(* Logix 5000 project; controller VET 1756-L62 rev 19.52; software revision 19.01; part 18 of 27 *)
(* tags used below, declared in another part *)
   dosif_struct : ALIAS FOR dosificador[1];
   dosificacion_interrumpida : BOOL;
   dosificando : BOOL;
   flags : DINT;
   idx_batch : DINT;
   idx_eqp1 : DINT;
   idx_eqp2 : DINT;
   idx_eqp3 : DINT;
   idx_eqp4 : DINT;
   idx_eqp5 : DINT;
   idx_ing : DINT;
   idx_tolv : DINT;   // Índice de Tolva
   resultado : ALIAS FOR dosif_struct.resultado;
   step_index : DINT;
   step_index_buffer : DINT;
   T : TIMER[15];
   _Eqp : Equipo[800];
   _Parametros_D : DINT[30];
   _Parametros_F : REAL[30];
   _reset_locales : DINT;
   Batch : batch[10];
   corriente : REAL[40];
   dosificador : dosif_struct[20];
   Dosificar_MID_01 : PHASE;
   fecha_plc : DINT;
   flujometro : flujometro[5];
   hora_plc : DINT;
   peso_tolva : REAL[80];
   SetDInt : DINT[500];
   TabBin : Bins_Setup;
   vdf : VDFS[20];
(* Dosificar_MID_01, continued *)

ROUTINE Holding   (* ladder *)
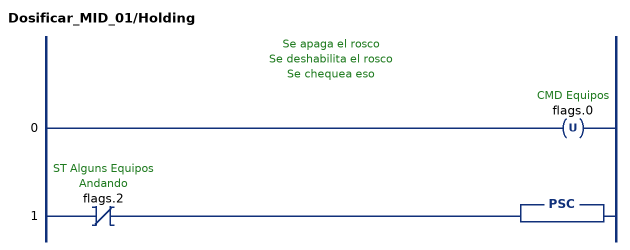
   // Se apaga el rosco
   // Se deshabilita el rosco
   // Se chequea eso
   0: OTU(flags.0);
   1: XIO(flags.2)PSC();
END_ROUTINE

ROUTINE preState   (* ladder *)
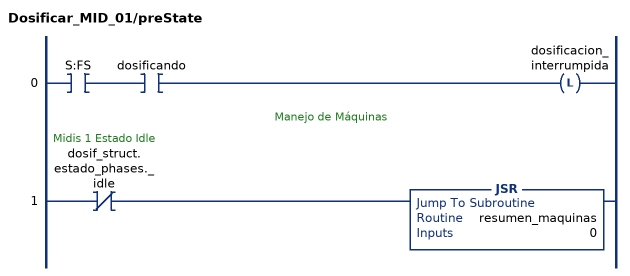
   0: XIC(S:FS)XIC(dosificando)OTL(dosificacion_interrumpida);
   // Manejo de Máquinas
   1: XIO(dosif_struct.estado_phases._idle)JSR(resumen_maquinas,0);
END_ROUTINE

ROUTINE Resetting   (* ladder *)
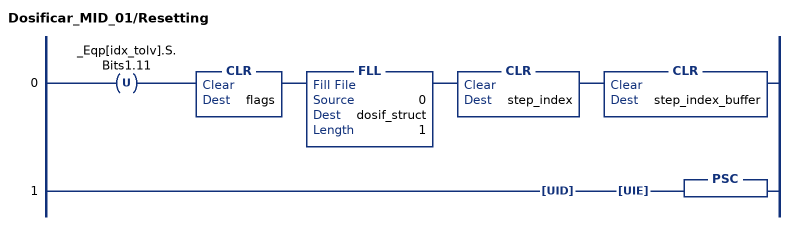
   0: OTU(_Eqp[idx_tolv].S.Bits1.11)CLR(flags)FLL(0,dosif_struct,1)CLR(step_index)CLR(step_index_buffer);
   1: UID()UIE()PSC();
END_ROUTINE

ROUTINE Restarting   (* ladder *)
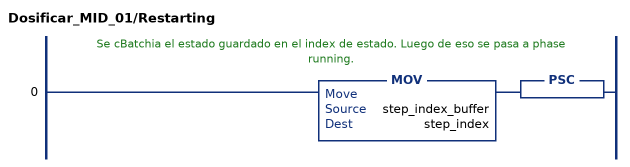
   // Se cBatchia el estado guardado en el index de estado. Luego de eso se pasa a phase running.
   0: MOV(step_index_buffer,step_index)PSC();
END_ROUTINE

ROUTINE resumen_maquinas   (* ladder *)
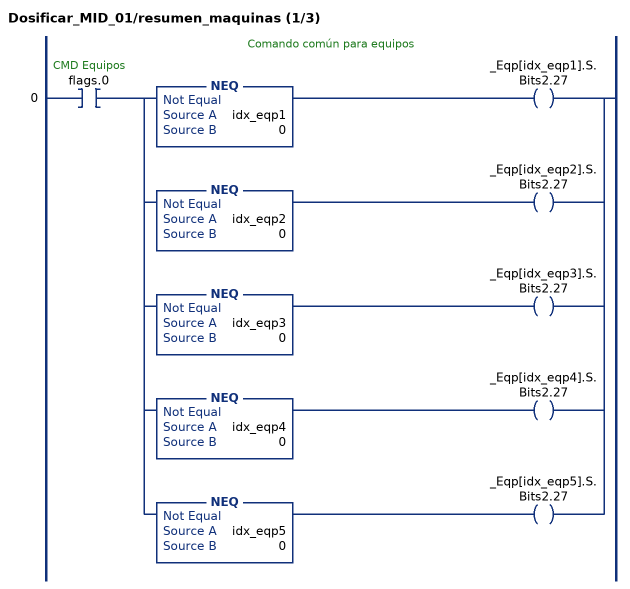
   // Comando común para equipos
   0: XIC(flags.0)[NEQ(idx_eqp1,0) OTE(_Eqp[idx_eqp1].S.Bits2.27) ,NEQ(idx_eqp2,0) OTE(_Eqp[idx_eqp2].S.Bits2.27) ,NEQ(idx_eqp3,0) OTE(_Eqp[idx_eqp3].S.Bits2.27) ,NEQ(idx_eqp4,0) OTE(_Eqp[idx_eqp4].S.Bits2.27) ,NEQ(idx_eqp5,0) OTE(_Eqp[idx_eqp5].S.Bits2.27) ];
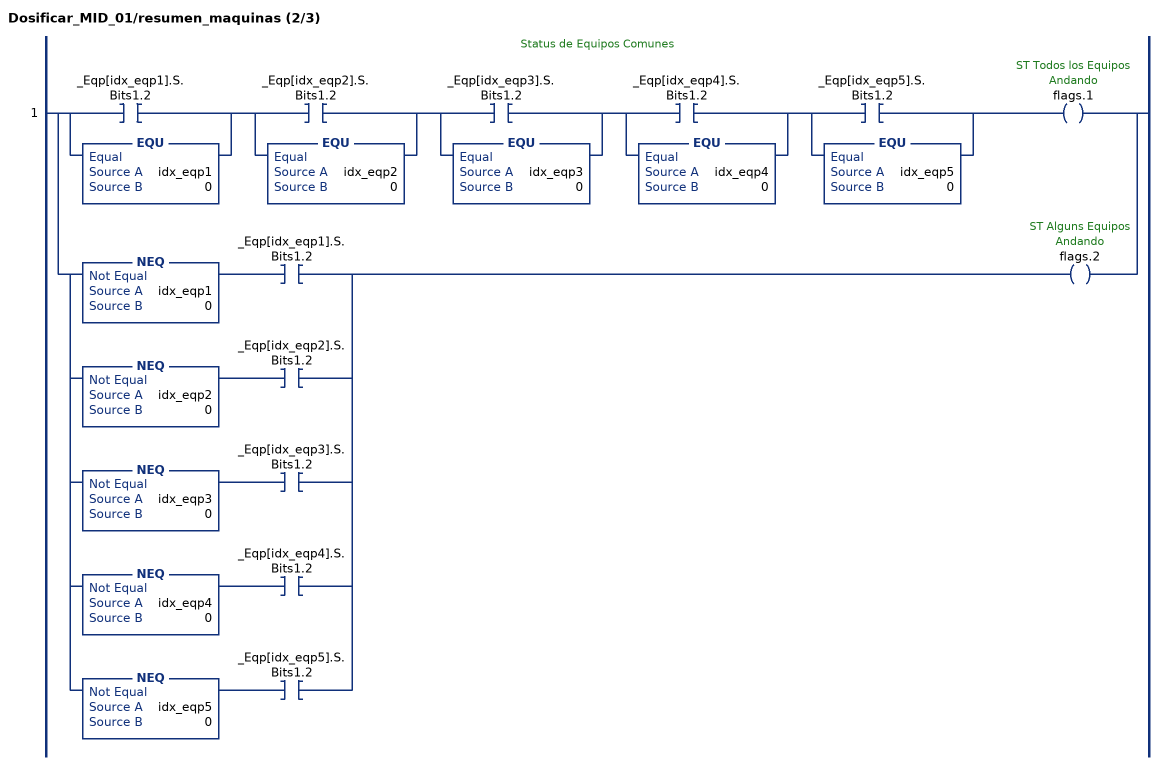
   // Status de Equipos Comunes
   1: [[XIC(_Eqp[idx_eqp1].S.Bits1.2) ,EQU(idx_eqp1,0) ] [XIC(_Eqp[idx_eqp2].S.Bits1.2) ,EQU(idx_eqp2,0) ] [XIC(_Eqp[idx_eqp3].S.Bits1.2) ,EQU(idx_eqp3,0) ] [XIC(_Eqp[idx_eqp4].S.Bits1.2) ,EQU(idx_eqp4,0) ] [XIC(_Eqp[idx_eqp5].S.Bits1.2) ,EQU(idx_eqp5,0) ] OTE(flags.1) ,[NEQ(idx_eqp1,0) XIC(_Eqp[idx_eqp1].S.Bits1.2) ,NEQ(idx_eqp2,0) XIC(_Eqp[idx_eqp2].S.Bits1.2) ,NEQ(idx_eqp3,0) XIC(_Eqp[idx_eqp3].S.Bits1.2) ,NEQ(idx_eqp4,0) XIC(_Eqp[idx_eqp4].S.Bits1.2) ,NEQ(idx_eqp5,0) XIC(_Eqp[idx_eqp5].S.Bits1.2) ] OTE(flags.2) ];
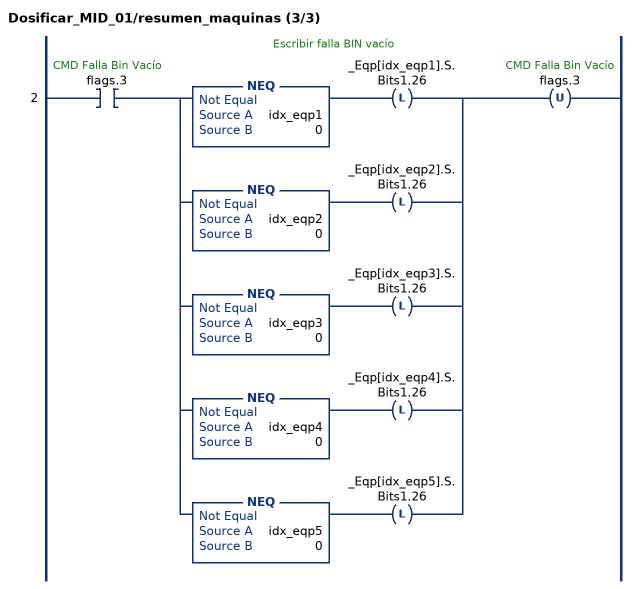
   // Escribir falla BIN vacío
   2: XIC(flags.3)[NEQ(idx_eqp1,0) OTL(_Eqp[idx_eqp1].S.Bits1.26) ,NEQ(idx_eqp2,0) OTL(_Eqp[idx_eqp2].S.Bits1.26) ,NEQ(idx_eqp3,0) OTL(_Eqp[idx_eqp3].S.Bits1.26) ,NEQ(idx_eqp4,0) OTL(_Eqp[idx_eqp4].S.Bits1.26) ,NEQ(idx_eqp5,0) OTL(_Eqp[idx_eqp5].S.Bits1.26) ]OTU(flags.3);
END_ROUTINE

ROUTINE Running   (* ladder *)
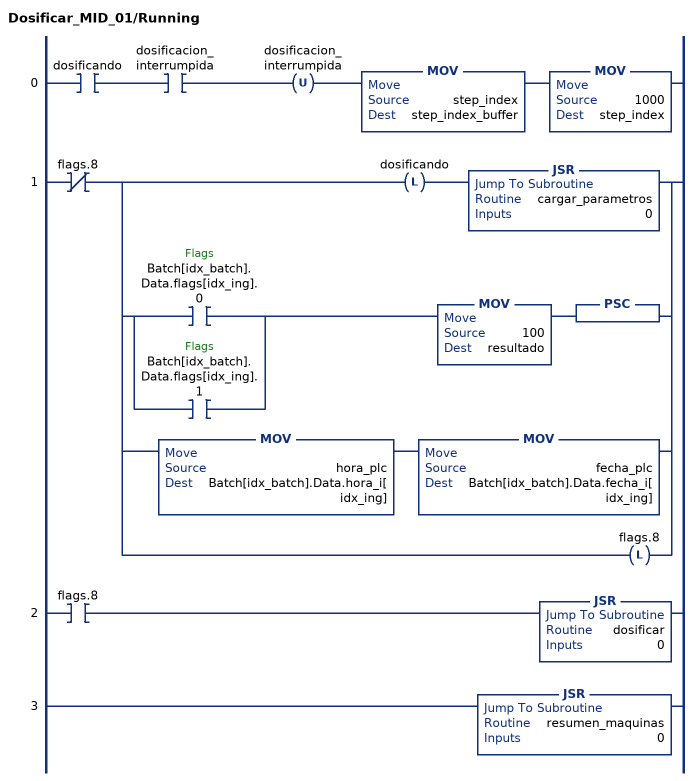
   0: XIC(dosificando)XIC(dosificacion_interrumpida)OTU(dosificacion_interrumpida)MOV(step_index,step_index_buffer)MOV(1000,step_index);
   1: XIO(flags.8)[OTL(dosificando) JSR(cargar_parametros,0) ,[[XIC(Batch[idx_batch].Data.flags[idx_ing].0) ,XIC(Batch[idx_batch].Data.flags[idx_ing].1) ] MOV(100,resultado) PSC() ,MOV(hora_plc,Batch[idx_batch].Data.hora_i[idx_ing]) MOV(fecha_plc,Batch[idx_batch].Data.fecha_i[idx_ing]) ] ,OTL(flags.8) ];
   2: XIC(flags.8)JSR(dosificar,0);
   3: JSR(resumen_maquinas,0);
END_ROUTINE
END_PROGRAM

PROGRAM Gestion_Dosificacion   (* main routine Main *)
VAR
   _fn1_auto : BOOL := 1;
   _fn1_ingrediente : DINT := 66;
   _fn1_lugar : DINT := 2;
   _fn1_ndx : DINT := 42;
   _fn1_prioridad : DINT;
   _fn1_tolva : DINT[2] := ([0] := 17);
   _fn2_batch_detalle : batch_detalle := (codigo[0] := 81, codigo[1] := 51, codigo[2] := 53, codigo[3] := 55, codigo[4] := 57, codigo[5] := 67, codigo[6] := 68, codigo[7] := 69, codigo[8] := 70, codigo[9] := 74, codigo[10] := 75, codigo[11] := 76, codigo[12] := 77, codigo[13] := 60, codigo[14] := 62, codigo[15] := 64, codigo[16] := 66, peso_f[0] := 70.0, peso_f[1] := 400.0, peso_f[2] := 350.0, peso_f[3] := 175.0, peso_f[4] := 225.0, peso_f[5] := 30.0, peso_f[6] := 25.0, peso_f[7] := 17.5, peso_f[8] := 17.5, peso_f[9] := 30.0, peso_f[10] := 5.0, peso_f[11] := 4.0, peso_f[12] := 4.0, peso_f[13] := 125.0, peso_f[14] := 125.0, peso_f[15] := 65.0, peso_f[16] := 65.0, tolva[0] := 38, tolva[2] := 4, tolva[3] := 10, tolva[4] := 12, tolva[5] := 18, tolva[6] := 19, tolva[7] := 20, tolva[8] := 21, tolva[9] := 26, tolva[10] := 27, tolva[11] := 28, tolva[12] := 29, tolva[13] := 7, tolva[14] := 9, tolva[15] := 15, tolva[16] := 17, lugar[0] := 6, lugar[2] := 1, lugar[3] := 1, lugar[4] := 1, lugar[5] := 3, lugar[6] := 3, lugar[7] := 3, lugar[8] := 3, lugar[9] := 4, lugar[10] := 4,
        lugar[11] := 4, lugar[12] := 4, lugar[13] := 2, lugar[14] := 2, lugar[15] := 2, lugar[16] := 2, flags[0] := 4, flags[2] := 4, flags[3] := 4, flags[4] := 4, flags[5] := 4, flags[6] := 4, flags[7] := 4, flags[8] := 4, flags[9] := 4, flags[10] := 4, flags[11] := 4, flags[12] := 4, flags[13] := 4, flags[14] := 4, flags[15] := 4, flags[16] := 4);
   _fn2_ndx : DINT := 17;
   _reset_local : ALIAS FOR _reset_locales.1;
   debug : BOOL;
   dsf_l : set_variables := (D[0] := 90748, D[1] := 60040, D[2] := 30001, T[0].PRE := 3500000, T[1].PRE := 60000, T[2].PRE := 30000, T[3].PRE := 3000, T[4].PRE := 40000, i0 := 40);   // Var. Dosificación Líquidos
        .I0   // Índice de Productos
        .D[10]   // Bits
        .D[11]   // Bits
        .D[12]   // Bits
        .D[10].0   // Manual 1 Listos
        .D[10].1   // Líquido 1 Listos
        .I1   // Índice de Productos listos
        .D[0]   // Tiempo Total en Mezcladora
        .D[1]   // Tiempo Mezcla
        .D[2]   // Tiempo Mezcla (Ingredientes)
        .D[11].0   // Opción de detención de Mezcladora
        .D[14]   // respuestas
        .D[13]   // mensajes
        .D[13].0   // Batch Abortado
        .D[14].0   // Aceptar
   dsf_s : set_variables := (D[0] := 1157052, D[13] := 1, T[0].PRE := 3000, T[1].PRE := 3000, T[2].PRE := 3000, T[3].PRE := 2975000, T[3].ACC := 1157052, T[3].EN := 1, T[3].TT := 1, T[7].PRE := 3000, i0 := 40, i2 := 6, i3 := 38, i4 := 5, i5 := 1);   // Var. Dosificación Sólidos
        .I2   // Índice interfaz IO dosif.
        .I0   // Índice Productos
        .D[0]   // Tiempo de Dosificación
        .D[10]   // Bits
        .D[11]   // Bits
        .D[12]   // Bits
        .D[10].0   // Macro-ingredientes Listos
        .D[10].1   // Midi-ingredientes Listos
        .D[10].2   // Micro-ingredientes 1 Listos
        .D[10].3   // Micro-ingredientes 2 Listos
        .I1   // Índice Productos Listos
        .I3   // Índice Peso Tolva
        .I4   // Índice Frec. VDF
        .D[11].0   // cmd. predescarga macros
        .D[11].1   // cmd. predescarga midis
        .D[11].2   // cmd. predescarga micros 1
        .D[11].3   // cmd. predescarga micros 2
        .T[4]   // Predescarga Macros
        .T[5]   // Predescarga Midis
        .T[6]   // Predescarga Micros 1
        .T[7]   // Predescarga Micros 2
        .D[14].1   // Devolver
        .D[13].0   // Dosificación Manual
        .D[14]   // respuestas
        .D[13]   // mensajes
        .I5   // Índice Productos Man (Conf)
        .D[14].0   // Aceptar
   estado : DINT[10] := ([0] := 8);
        [0]   // E. Gestión Sólidos
        [1]   // E. Gestión MAC 01
        [4]   // E. Gestión MIC 02
        [2]   // E. Gestión MID 01
        [3]   // E. Gestión MIC 01
        [5]   // E. G. Desc. Sol.
        [6]   // E. Gestión Líquidos
        [7]   // E. Gestión Transporte
END_VAR

ROUTINE _fn1_buscar_1_ingrediente   (* ladder *)
// Búsqueda de 1 ingrediente
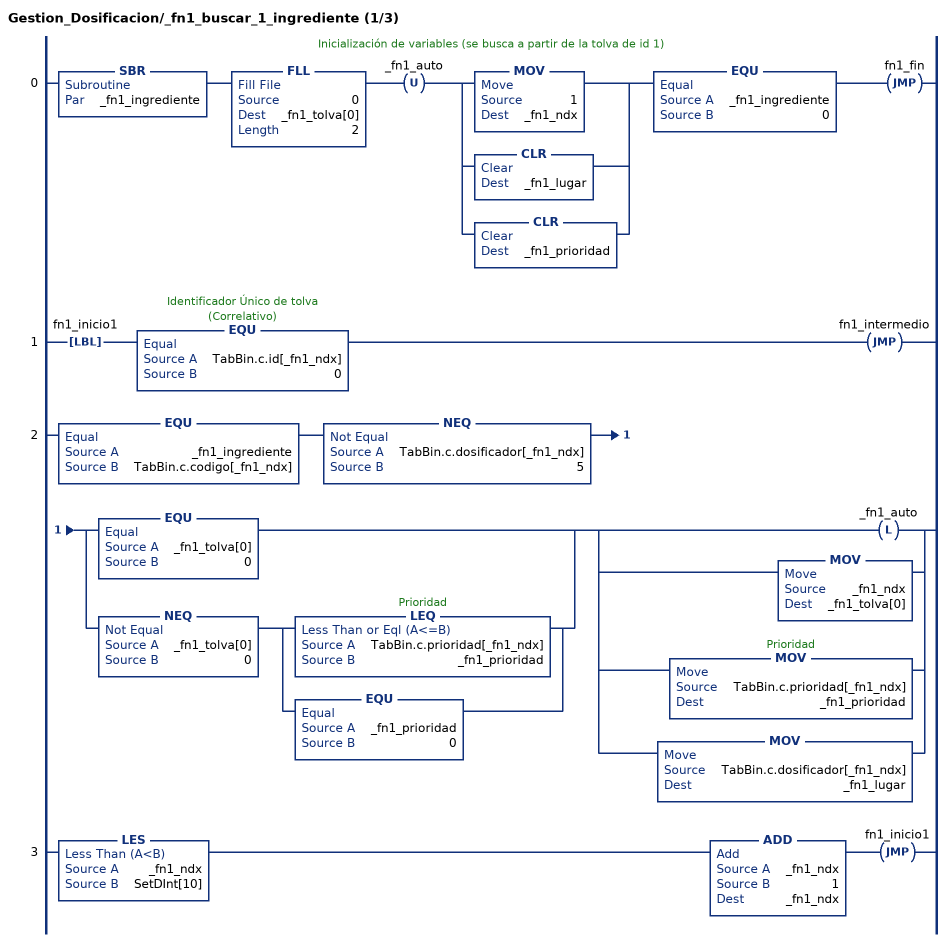
   // Inicialización de variables (se busca a partir de la tolva de id 1)
   0: SBR(_fn1_ingrediente)FLL(0,_fn1_tolva[0],2)OTU(_fn1_auto)[MOV(1,_fn1_ndx) ,CLR(_fn1_lugar) ,CLR(_fn1_prioridad) ]EQU(_fn1_ingrediente,0)JMP(fn1_fin);
   1: LBL(fn1_inicio1)EQU(TabBin.c.id[_fn1_ndx],0)JMP(fn1_intermedio);
   2: EQU(_fn1_ingrediente,TabBin.c.codigo[_fn1_ndx])NEQ(TabBin.c.dosificador[_fn1_ndx],5)[EQU(_fn1_tolva[0],0) ,NEQ(_fn1_tolva[0],0) [LEQ(TabBin.c.prioridad[_fn1_ndx],_fn1_prioridad) ,EQU(_fn1_prioridad,0) ] ][OTL(_fn1_auto) ,MOV(_fn1_ndx,_fn1_tolva[0]) ,MOV(TabBin.c.prioridad[_fn1_ndx],_fn1_prioridad) ,MOV(TabBin.c.dosificador[_fn1_ndx],_fn1_lugar) ];
   3: LES(_fn1_ndx,SetDInt[10])ADD(_fn1_ndx,1,_fn1_ndx)JMP(fn1_inicio1);
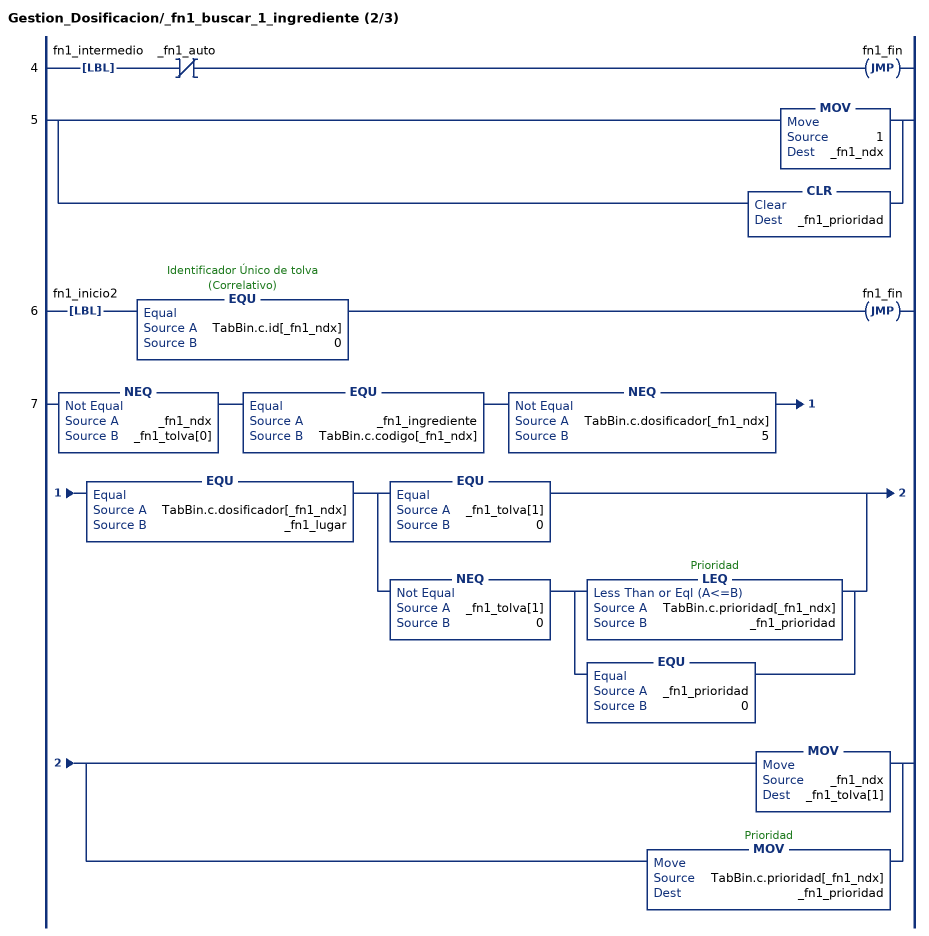
   4: LBL(fn1_intermedio)XIO(_fn1_auto)JMP(fn1_fin);
   5: [MOV(1,_fn1_ndx) ,CLR(_fn1_prioridad) ];
   6: LBL(fn1_inicio2)EQU(TabBin.c.id[_fn1_ndx],0)JMP(fn1_fin);
   7: NEQ(_fn1_ndx,_fn1_tolva[0])EQU(_fn1_ingrediente,TabBin.c.codigo[_fn1_ndx])NEQ(TabBin.c.dosificador[_fn1_ndx],5)EQU(TabBin.c.dosificador[_fn1_ndx],_fn1_lugar)[EQU(_fn1_tolva[1],0) ,NEQ(_fn1_tolva[1],0) [LEQ(TabBin.c.prioridad[_fn1_ndx],_fn1_prioridad) ,EQU(_fn1_prioridad,0) ] ][MOV(_fn1_ndx,_fn1_tolva[1]) ,MOV(TabBin.c.prioridad[_fn1_ndx],_fn1_prioridad) ];
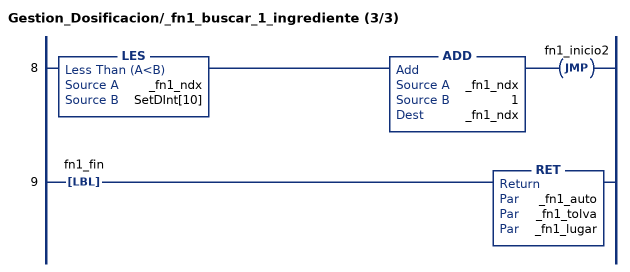
   8: LES(_fn1_ndx,SetDInt[10])ADD(_fn1_ndx,1,_fn1_ndx)JMP(fn1_inicio2);
   9: LBL(fn1_fin)RET(_fn1_auto,_fn1_tolva,_fn1_lugar);
END_ROUTINE

ROUTINE _fn2_buscar_ingredientes   (* ladder *)
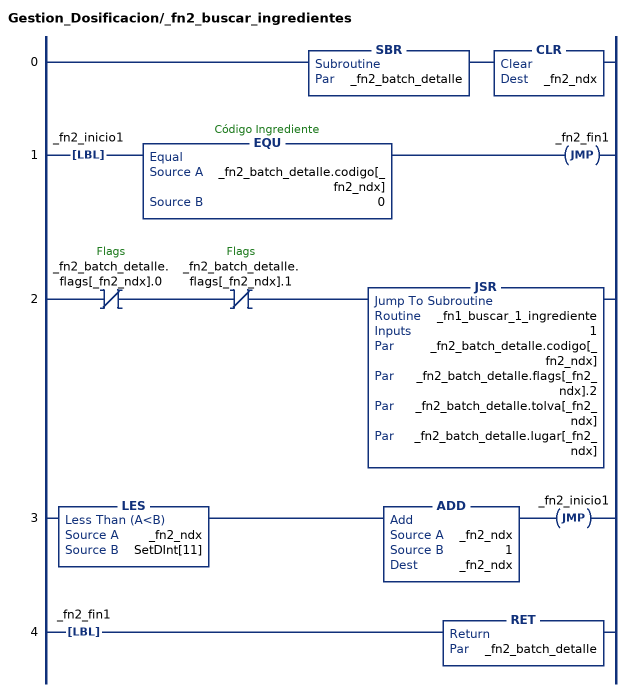
   0: SBR(_fn2_batch_detalle)CLR(_fn2_ndx);
   1: LBL(_fn2_inicio1)EQU(_fn2_batch_detalle.codigo[_fn2_ndx],0)JMP(_fn2_fin1);
   2: XIO(_fn2_batch_detalle.flags[_fn2_ndx].0)XIO(_fn2_batch_detalle.flags[_fn2_ndx].1)JSR(_fn1_buscar_1_ingrediente,1,_fn2_batch_detalle.codigo[_fn2_ndx],_fn2_batch_detalle.flags[_fn2_ndx].2,_fn2_batch_detalle.tolva[_fn2_ndx],_fn2_batch_detalle.lugar[_fn2_ndx]);
   3: LES(_fn2_ndx,SetDInt[11])ADD(_fn2_ndx,1,_fn2_ndx)JMP(_fn2_inicio1);
   4: LBL(_fn2_fin1)RET(_fn2_batch_detalle);
END_ROUTINE

ROUTINE Gestion_Descargas_Solidos   (* ladder *)
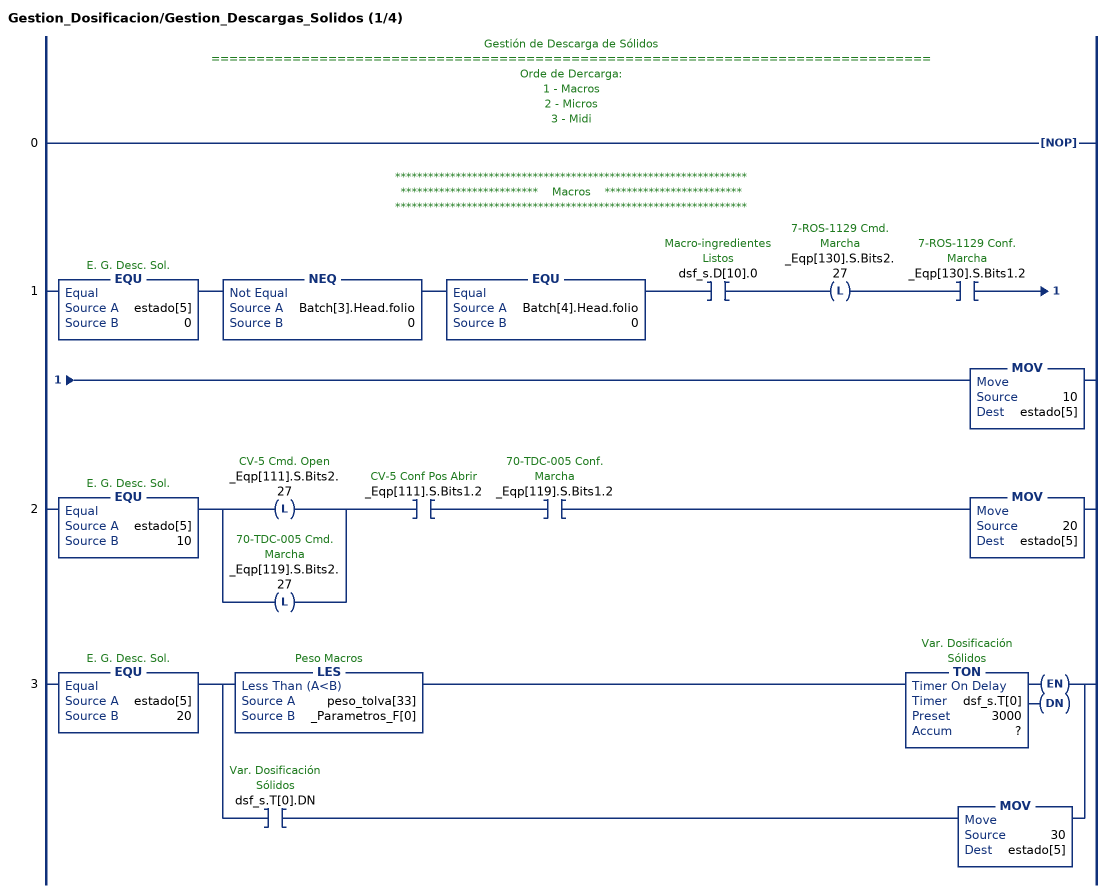
   // Gestión de Descarga de Sólidos
   // ================================================================================
   // Orde de Dercarga:
   // 1 - Macros
   // 2 - Micros
   // 3 - Midi
   0: NOP();
   // ****************************************************************
   // *************************    Macros    *************************
   // ****************************************************************
   1: EQU(estado[5],0)NEQ(Batch[3].Head.folio,0)EQU(Batch[4].Head.folio,0)XIC(dsf_s.D[10].0)OTL(_Eqp[130].S.Bits2.27)XIC(_Eqp[130].S.Bits1.2)MOV(10,estado[5]);
   2: EQU(estado[5],10)[OTL(_Eqp[111].S.Bits2.27) ,OTL(_Eqp[119].S.Bits2.27) ]XIC(_Eqp[111].S.Bits1.2)XIC(_Eqp[119].S.Bits1.2)MOV(20,estado[5]);
   3: EQU(estado[5],20)[LES(peso_tolva[33],_Parametros_F[0]) TON(dsf_s.T[0],?,?) ,XIC(dsf_s.T[0].DN) MOV(30,estado[5]) ];
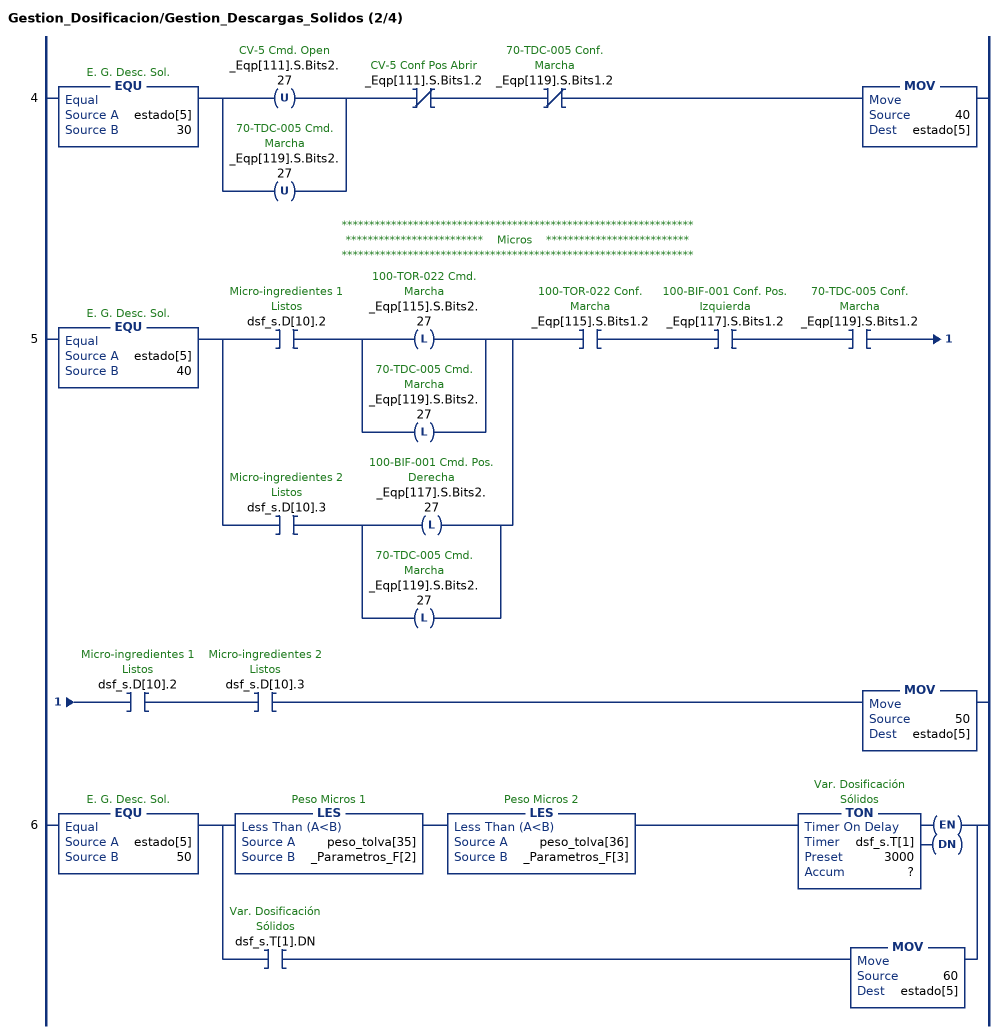
   4: EQU(estado[5],30)[OTU(_Eqp[111].S.Bits2.27) ,OTU(_Eqp[119].S.Bits2.27) ]XIO(_Eqp[111].S.Bits1.2)XIO(_Eqp[119].S.Bits1.2)MOV(40,estado[5]);
   // ****************************************************************
   // *************************    Micros    **************************
   // ****************************************************************
   5: EQU(estado[5],40)[XIC(dsf_s.D[10].2) [OTL(_Eqp[115].S.Bits2.27) ,OTL(_Eqp[119].S.Bits2.27) ] ,XIC(dsf_s.D[10].3) [OTL(_Eqp[117].S.Bits2.27) ,OTL(_Eqp[119].S.Bits2.27) ] ]XIC(_Eqp[115].S.Bits1.2)XIC(_Eqp[117].S.Bits1.2)XIC(_Eqp[119].S.Bits1.2)XIC(dsf_s.D[10].2)XIC(dsf_s.D[10].3)MOV(50,estado[5]);
   6: EQU(estado[5],50)[LES(peso_tolva[35],_Parametros_F[2]) LES(peso_tolva[36],_Parametros_F[3]) TON(dsf_s.T[1],?,?) ,XIC(dsf_s.T[1].DN) MOV(60,estado[5]) ];
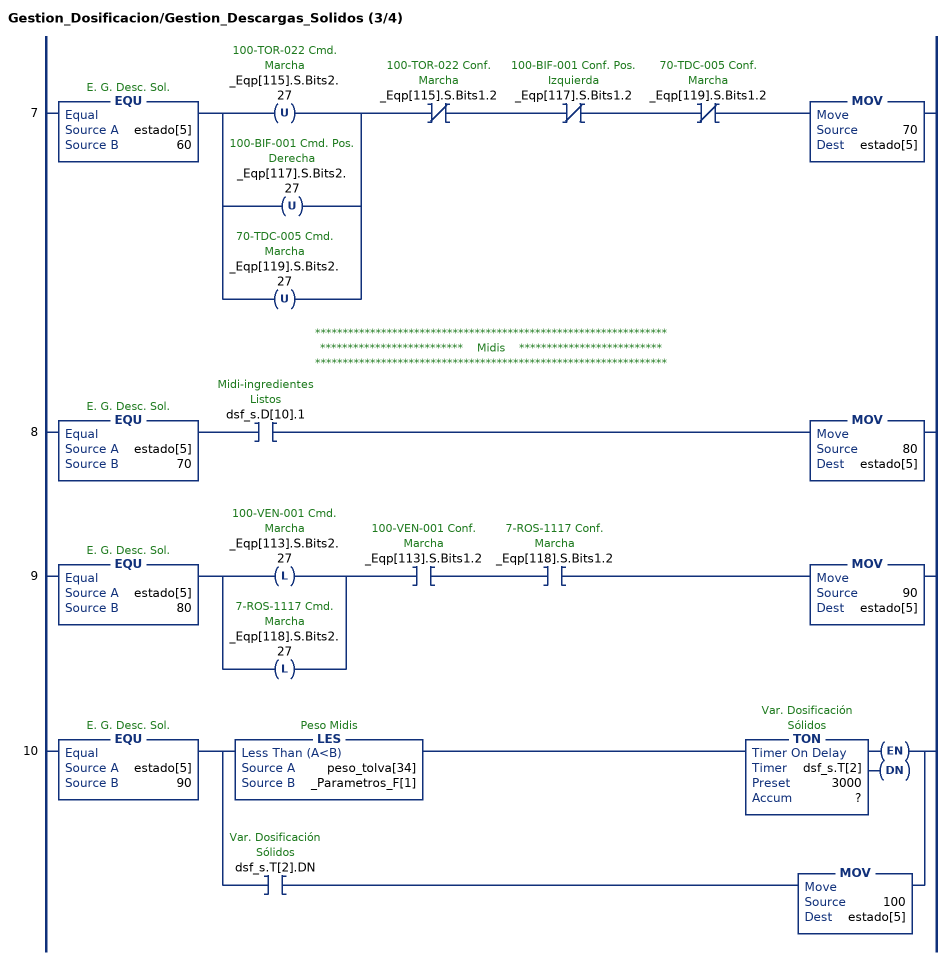
   7: EQU(estado[5],60)[OTU(_Eqp[115].S.Bits2.27) ,OTU(_Eqp[117].S.Bits2.27) ,OTU(_Eqp[119].S.Bits2.27) ]XIO(_Eqp[115].S.Bits1.2)XIO(_Eqp[117].S.Bits1.2)XIO(_Eqp[119].S.Bits1.2)MOV(70,estado[5]);
   // ****************************************************************
   // **************************    Midis    **************************
   // ****************************************************************
   8: EQU(estado[5],70)XIC(dsf_s.D[10].1)MOV(80,estado[5]);
   9: EQU(estado[5],80)[OTL(_Eqp[113].S.Bits2.27) ,OTL(_Eqp[118].S.Bits2.27) ]XIC(_Eqp[113].S.Bits1.2)XIC(_Eqp[118].S.Bits1.2)MOV(90,estado[5]);
   10: EQU(estado[5],90)[LES(peso_tolva[34],_Parametros_F[1]) TON(dsf_s.T[2],?,?) ,XIC(dsf_s.T[2].DN) MOV(100,estado[5]) ];
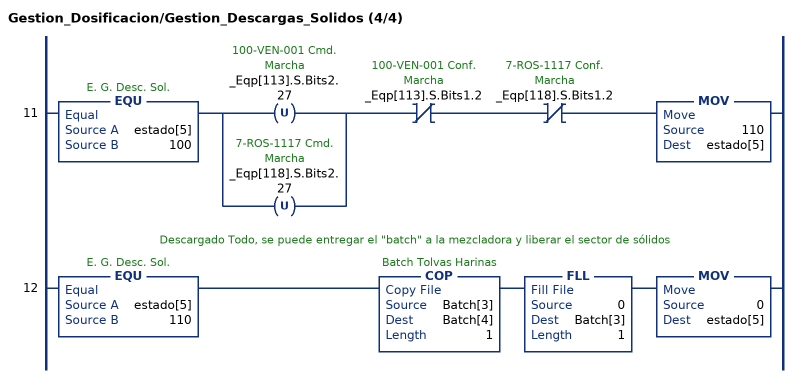
   11: EQU(estado[5],100)[OTU(_Eqp[113].S.Bits2.27) ,OTU(_Eqp[118].S.Bits2.27) ]XIO(_Eqp[113].S.Bits1.2)XIO(_Eqp[118].S.Bits1.2)MOV(110,estado[5]);
   // Descargado Todo, se puede entregar el "batch" a la mezcladora y liberar el sector de sólidos
   12: EQU(estado[5],110)COP(Batch[3],Batch[4],1)FLL(0,Batch[3],1)MOV(0,estado[5]);
END_ROUTINE

ROUTINE Gestion_Liquidos   (* ladder *)
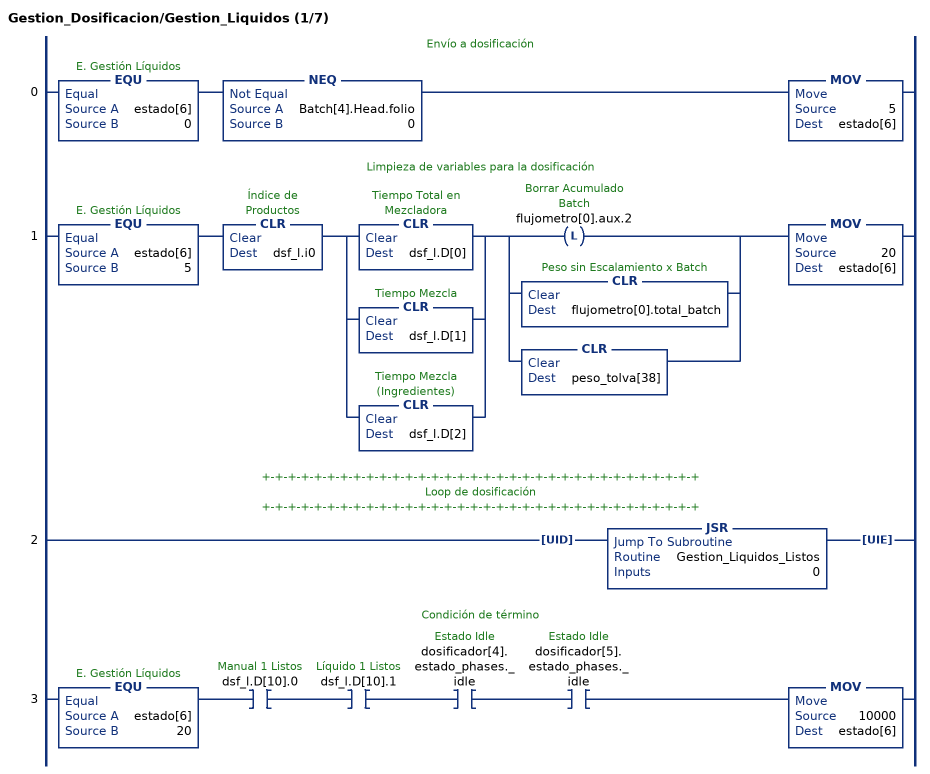
   // Envío a dosificación
   0: EQU(estado[6],0)NEQ(Batch[4].Head.folio,0)MOV(5,estado[6]);
   // Limpieza de variables para la dosificación
   1: EQU(estado[6],5)CLR(dsf_l.i0)[CLR(dsf_l.D[0]) ,CLR(dsf_l.D[1]) ,CLR(dsf_l.D[2]) ][OTL(flujometro[0].aux.2) ,CLR(flujometro[0].total_batch) ,CLR(peso_tolva[38]) ]MOV(20,estado[6]);
   // +-+-+-+-+-+-+-+-+-+-+-+-+-+-+-+-+-+-+-+-+-+-+-+-+-+-+-+-+-+-+-+-+-+
   // Loop de dosificación
   // +-+-+-+-+-+-+-+-+-+-+-+-+-+-+-+-+-+-+-+-+-+-+-+-+-+-+-+-+-+-+-+-+-+
   2: UID()JSR(Gestion_Liquidos_Listos,0)UIE();
   // Condición de término
   3: EQU(estado[6],20)XIC(dsf_l.D[10].0)XIC(dsf_l.D[10].1)XIC(dosificador[4].estado_phases._idle)XIC(dosificador[5].estado_phases._idle)MOV(10000,estado[6]);
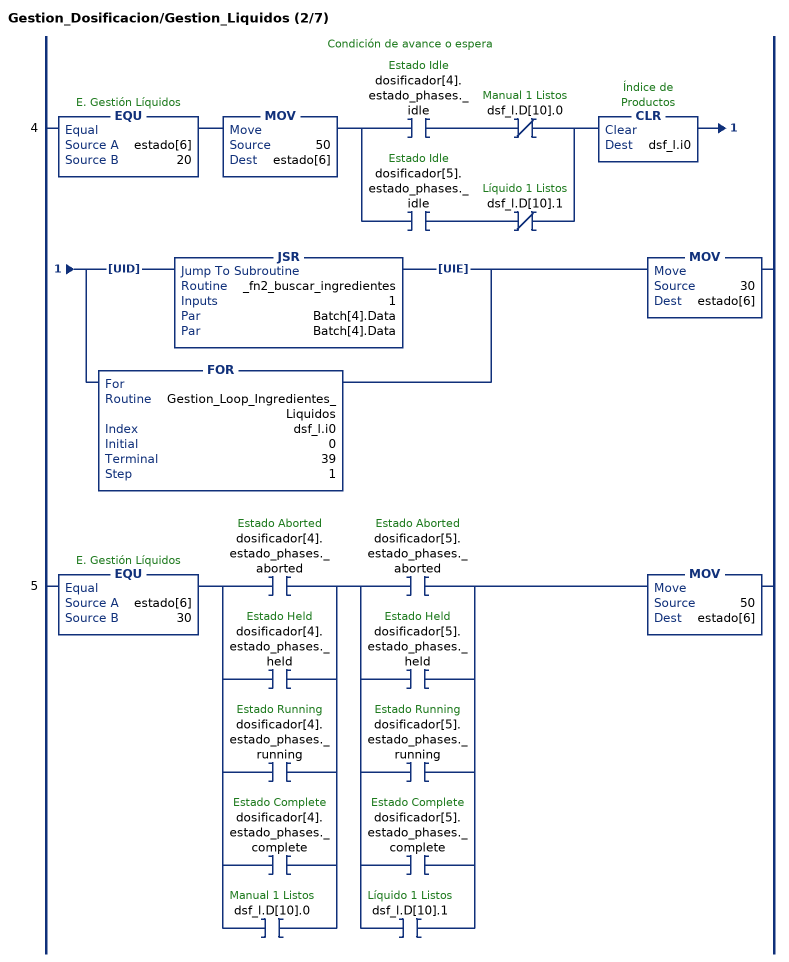
   // Condición de avance o espera
   4: EQU(estado[6],20)MOV(50,estado[6])[XIC(dosificador[4].estado_phases._idle) XIO(dsf_l.D[10].0) ,XIC(dosificador[5].estado_phases._idle) XIO(dsf_l.D[10].1) ]CLR(dsf_l.i0)[UID() JSR(_fn2_buscar_ingredientes,1,Batch[4].Data,Batch[4].Data) UIE() ,FOR(Gestion_Loop_Ingredientes_Liquidos,dsf_l.i0,0,39,1) ]MOV(30,estado[6]);
   5: EQU(estado[6],30)[XIC(dosificador[4].estado_phases._aborted) ,XIC(dosificador[4].estado_phases._held) ,XIC(dosificador[4].estado_phases._running) ,XIC(dosificador[4].estado_phases._complete) ,XIC(dsf_l.D[10].0) ][XIC(dosificador[5].estado_phases._aborted) ,XIC(dosificador[5].estado_phases._held) ,XIC(dosificador[5].estado_phases._running) ,XIC(dosificador[5].estado_phases._complete) ,XIC(dsf_l.D[10].1) ]MOV(50,estado[6]);
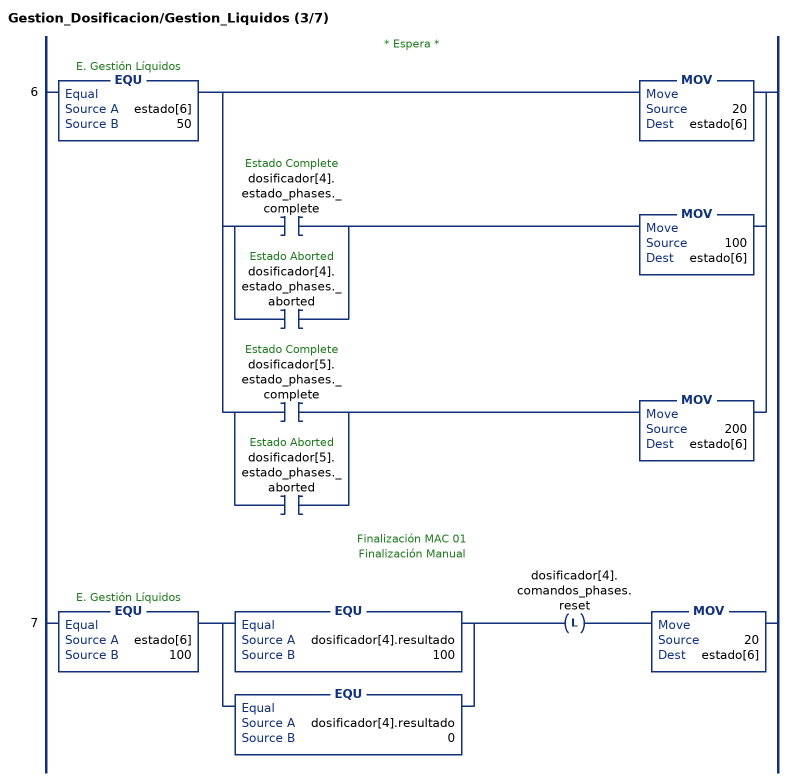
   // * Espera *
   6: EQU(estado[6],50)[MOV(20,estado[6]) ,[XIC(dosificador[4].estado_phases._complete) ,XIC(dosificador[4].estado_phases._aborted) ] MOV(100,estado[6]) ,[XIC(dosificador[5].estado_phases._complete) ,XIC(dosificador[5].estado_phases._aborted) ] MOV(200,estado[6]) ];
   // Finalización MAC 01
   // Finalización Manual
   7: EQU(estado[6],100)[EQU(dosificador[4].resultado,100) ,EQU(dosificador[4].resultado,0) ]OTL(dosificador[4].comandos_phases.reset)MOV(20,estado[6]);
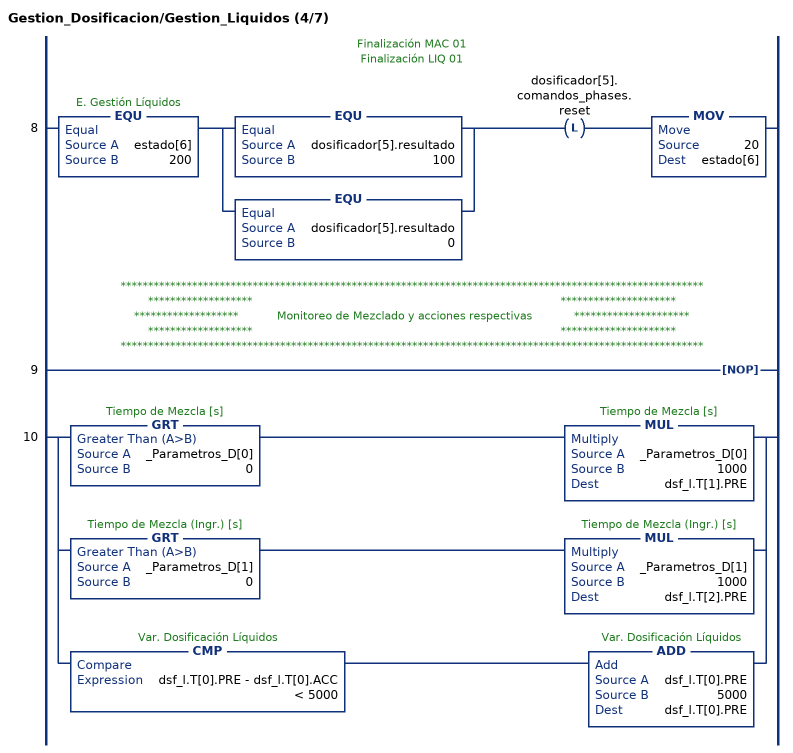
   // Finalización MAC 01
   // Finalización LIQ 01
   8: EQU(estado[6],200)[EQU(dosificador[5].resultado,100) ,EQU(dosificador[5].resultado,0) ]OTL(dosificador[5].comandos_phases.reset)MOV(20,estado[6]);
   // **********************************************************************************************************
   // *******************                                                                                        *********************
   // *******************           Monitoreo de Mezclado y acciones respectivas            *********************
   // *******************                                                                                        *********************
   // **********************************************************************************************************
   9: NOP();
   10: [GRT(_Parametros_D[0],0) MUL(_Parametros_D[0],1000,dsf_l.T[1].PRE) ,GRT(_Parametros_D[1],0) MUL(_Parametros_D[1],1000,dsf_l.T[2].PRE) ,CMP(dsf_l.T[0].PRE - dsf_l.T[0].ACC < 5000) ADD(dsf_l.T[0].PRE,5000,dsf_l.T[0].PRE) ];
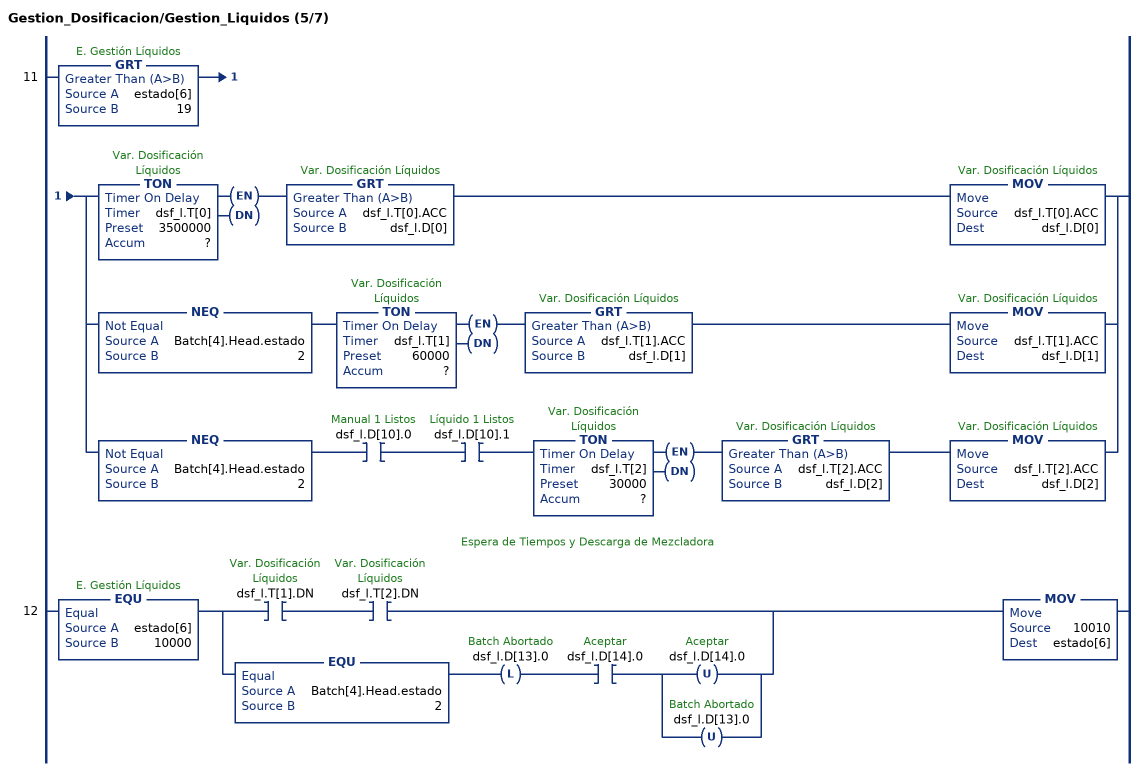
   11: GRT(estado[6],19)[TON(dsf_l.T[0],?,?) GRT(dsf_l.T[0].ACC,dsf_l.D[0]) MOV(dsf_l.T[0].ACC,dsf_l.D[0]) ,NEQ(Batch[4].Head.estado,2) TON(dsf_l.T[1],?,?) GRT(dsf_l.T[1].ACC,dsf_l.D[1]) MOV(dsf_l.T[1].ACC,dsf_l.D[1]) ,NEQ(Batch[4].Head.estado,2) XIC(dsf_l.D[10].0) XIC(dsf_l.D[10].1) TON(dsf_l.T[2],?,?) GRT(dsf_l.T[2].ACC,dsf_l.D[2]) MOV(dsf_l.T[2].ACC,dsf_l.D[2]) ];
   // Espera de Tiempos y Descarga de Mezcladora
   12: EQU(estado[6],10000)[XIC(dsf_l.T[1].DN) XIC(dsf_l.T[2].DN) ,EQU(Batch[4].Head.estado,2) OTL(dsf_l.D[13].0) XIC(dsf_l.D[14].0) [OTU(dsf_l.D[14].0) ,OTU(dsf_l.D[13].0) ] ]MOV(10010,estado[6]);
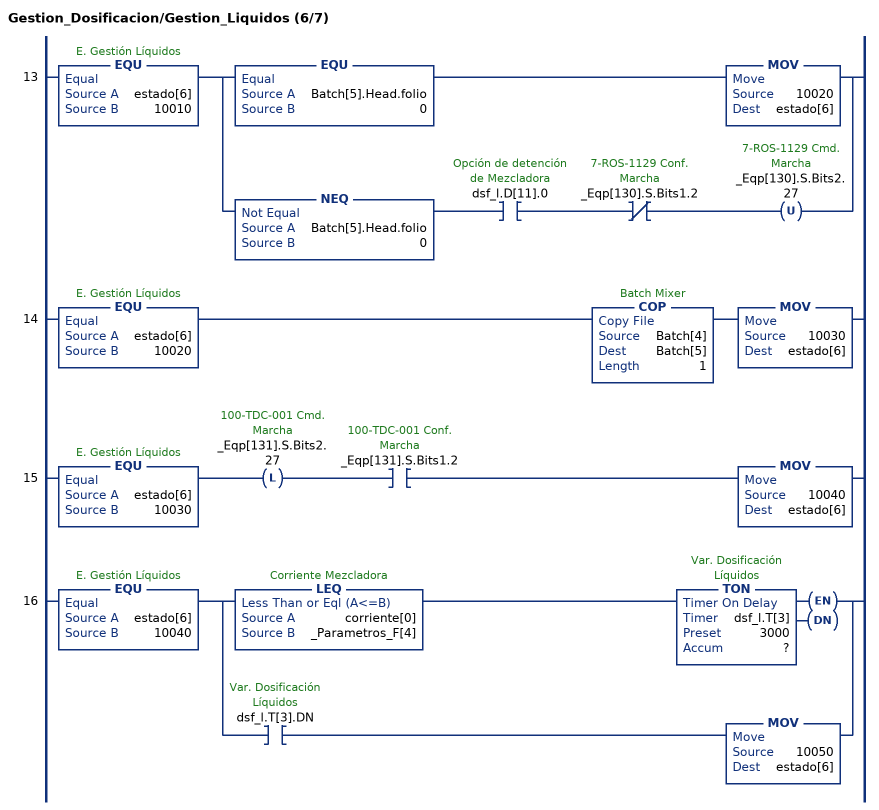
   13: EQU(estado[6],10010)[EQU(Batch[5].Head.folio,0) MOV(10020,estado[6]) ,NEQ(Batch[5].Head.folio,0) XIC(dsf_l.D[11].0) XIO(_Eqp[130].S.Bits1.2) OTU(_Eqp[130].S.Bits2.27) ];
   14: EQU(estado[6],10020)COP(Batch[4],Batch[5],1)MOV(10030,estado[6]);
   15: EQU(estado[6],10030)OTL(_Eqp[131].S.Bits2.27)XIC(_Eqp[131].S.Bits1.2)MOV(10040,estado[6]);
   16: EQU(estado[6],10040)[LEQ(corriente[0],_Parametros_F[4]) TON(dsf_l.T[3],?,?) ,XIC(dsf_l.T[3].DN) MOV(10050,estado[6]) ];
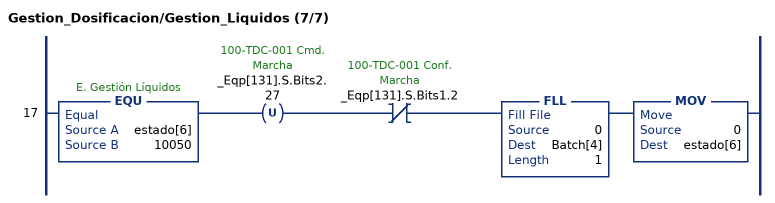
   17: EQU(estado[6],10050)OTU(_Eqp[131].S.Bits2.27)XIO(_Eqp[131].S.Bits1.2)FLL(0,Batch[4],1)MOV(0,estado[6]);
END_ROUTINE
